// TIA Portal V20 export
// export: Created 2026-04-11T06:02:30.0616572Z, ExportSetting WithDefaults, DisplayName Totally Integrated Automation Portal, DisplayVersion V20, DisplayName TIA Portal Openness, DisplayVersion V20, DisplayName TIA Portal Version Control Interface, DisplayVersion V20, DisplayName STEP 7 Professional, DisplayVersion V20, DisplayName STEP 7 Safety, DisplayVersion V20, DisplayName WinCC Basic/Comfort/Advanced, DisplayVersion V20, DisplayName WinCC Unified, DisplayVersion V20
TYPE "udtError_PID_Compact"
// stored: IsFailsafeCompliant false
   STRUCT
      InputOutOfRange { ExternalWritable := 'False'} : Bool;   // Input value is out of the configured range
      InputPERInvalid { ExternalWritable := 'False'} : Bool;   // InputPER value is invalid
      ValueOscillationFailed { ExternalWritable := 'False'} : Bool;   // Fine tuning - process value oscillation could not be maintained
      ProcessValueCloseToSetPoint { ExternalWritable := 'False'} : Bool;   // Pre-tuning - process value is too close to set point
      SetPointChangedDuringTuning { ExternalWritable := 'False'} : Bool;   // PID set point was changed during tuning
      PretuningDuringFineTuning { ExternalWritable := 'False'} : Bool;   // Pre-tuning not allowed while fine tuning is active
      InvalidOutputValueLimits { ExternalWritable := 'False'} : Bool;   // Pre-tuning - invalid configuration of output value limits
      InvalidFineTuningParameter { ExternalWritable := 'False'} : Bool;   // Fine tuning - error occurred causing invalid parameters
      InputInvalidFormat { ExternalWritable := 'False'} : Bool;   // Input value has an invalid number format
      OutputCalculationError { ExternalWritable := 'False'} : Bool;   // Output value calculation error ocurred
      SamplingTimeError { ExternalWritable := 'False'} : Bool;   // PID_Compact not called within sampling time of cyclic interrupt OB
      SetPointInvalidFormat { ExternalWritable := 'False'} : Bool;   // Set point value has an invalid number format
      ManualInvalidFormat { ExternalWritable := 'False'} : Bool;   // Manual value has an invalid number format
      SubstituteOutputInvalidFormat { ExternalWritable := 'False'} : Bool;   // Substitute output value has an invalid number format
      DisturbanceInvalidFormat { ExternalWritable := 'False'} : Bool;   // Disturbance value has an invlaid number format
   END_STRUCT;
END_TYPE
